// TIA Portal V19 export
DATA_BLOCK "InstCallGlobal"   // DB25
// stored: InstanceOfName CallGlobal, InstanceOfType FB
"CallGlobal"
   // VAR
   //    statClockSysMemOld { ExternalWritable := 'False'} : Byte;
   //    instLAF_PowerOnOff { ExternalWritable := 'False'} : "LAF_PowerOnOff";
   //    instLAF_ClockGen { ExternalWritable := 'False'} : "LAF_ClockGenerator";
   //    instLSNTP_Server { ExternalWritable := 'False'} : "LSNTP_Server";
   //    instLAF_SpecialFunctionsManager { S7_SetPoint := 'True'} : "LAF_SpecialFunctionsManager";
   // END_VAR
BEGIN
END_DATA_BLOCK
